// Core §3.8b/§3.10.2 — one editable value a module has registered about itself.
// The module declares it once at Setup; the framework then both PUBLISHES the
// capability (M_AppendConfig) and APPLIES writes to it (M_ApplyConfigWrite) from
// this single record, so the metadata a client validates against and the target
// the PLC writes can never drift apart (§1.1 O1/O9).
//
// pTarget is a pointer held in ordinary VAR — never inside a persistent
// declaration, where TwinCAT would retain an address that means nothing after a
// restart (TC3 §3.8b).
TYPE ST_ConfigWriteDef :
STRUCT
    Key           : STRING(160);  // §3.10.2 WriteKey — the mutation identity
    Item          : STRING(255);  // browse/display fragment; never the write identity
    Revision      : UDINT;        // non-zero; bump when the value's meaning changes
    Kind          : E_ConfigKind;
    ValueType     : E_ConfigValueType;
    Storage       : E_ConfigStorage;
    pTarget       : PVOID;
    RequiresReady : BOOL;         // write refused unless the owning root is READY
    HasMinimum    : BOOL;
    HasMaximum    : BOOL;
    Minimum       : LREAL;
    Maximum       : LREAL;
    Unit          : STRING(16);
    LabelKey      : STRING(160);
    MaxLength     : UINT;         // AS_STRING only: the target's declared capacity
    EnumDomain    : STRING(255);  // pipe-separated exact accepted values ('' = none)
    // §3.8c teach capture. The live source lives on the SAME record as the value
    // it writes, so a capture cannot reach a field that is not independently
    // editable - the back door §3.8c(a) forbids is structurally impossible here
    // rather than prevented by a check somebody could forget.
    // 0 = this value offers no capture, which is the default and most values.
    pCapture       : PVOID;
    CaptureStorage : E_ConfigStorage;   // how to READ the source (may differ from Storage)
    // §3.8d - the access axis. '' + NONE/NONE is the built-in class, which is
    // exactly the behaviour before data classes existed.
    ClassId       : STRING(40);
    MinReadLevel  : E_AccessLevel;
    MinWriteLevel : E_AccessLevel;
END_STRUCT
END_TYPE

(* stored: Version 1.1.0.1, ProductVersion 3.1.4024.12
   DUT ST_ConfigWriteDef: Id {7c418d55-9b02-4e37-8a6d-14f9b2e05c73} *)
